FUNCTION yGetActiveSection : BYTE
VAR_IN_OUT
	yActiveSections		: BYTE;
END_VAR
VAR
	ySectionChecked		: BYTE;
END_VAR

yGetActiveSection := 0;
WHILE TRUE DO
	ySectionChecked := LREAL_TO_BYTE(EXPT(2,yGetActiveSection));
	yGetActiveSection := yGetActiveSection + 1;
	IF (yActiveSections AND ySectionChecked) > 0 THEN
		(* Section found *)
		yActiveSections := yActiveSections - (yActiveSections AND ySectionChecked);
		EXIT;
	ELSIF yActiveSections = 0 THEN
		yGetActiveSection := 0;
		EXIT;
	END_IF
END_WHILE;

END_FUNCTION

(* stored: Version 1.1.0.1, ProductVersion 3.1.4022.12
   POU yGetActiveSection: Id {84f81a9d-340f-487e-b243-5f2b1027cd08}, SpecialFunc None *)
